FUNCTION_BLOCK FB_UMC EXTENDS FB_CtrlBase
VAR_INPUT
	In_uinStatus				: UINT;
	In_intMotorActualSpeed		: INT;
	In_uinMotorSetSpeed			: UINT;
	In_strNetId					: AMSNETID;
	In_uintPort					: WORD;
	In_uinECATState				: UINT;
	In_bolEmoOk					: BOOL;
END_VAR
VAR_OUTPUT
	Out_uinControl      	: UINT;
	Out_uinSpeedSetpoint	: UINT;
END_VAR
VAR
	/// Specific interface struct for public access
	SIf					: T_Ctrl_SIf_UMC;
	In_unStatus			: U_UMC_Lenze_Status;
	Out_unControl		: U_UMC_Lenze_Control;
	arTurnDirection		: ARRAY[0..MAX_E_TURN_DIRECTION] OF BOOL;
	fbPulse				: TC2_STANDARD.TP;
END_VAR
VAR CONSTANT
	cLEFT				: BOOL := TRUE;
	cRIGHT				: BOOL := FALSE;

	cEtherCAT_OP_MODE		: UINT := 16#0008;
	cEtherCAT_MODE_MASK		: UINT := 16#000F;
END_VAR

(*__________________________________________________________________________________________________
¦	
¦	Vistaprint Schweiz GmbH
¦	CH - 8401 Winterthur
¦
¦	www.vistaprint.ch - info@vistaprint.ch
¦___________________________________________________________________________________________________

Function desription:
Lenze Motor implementation. 


History:
Version		Date			Author		Comment
---------------------------------------------------------------------------------------------------
0.00.1		09.07.2013		PC			Start history
0.00.2		04.02.2014		AVM/MRU		Simulation mode
										cCMD_LEFT / cCMD_RIGHT added in FB_init / getCmdState

___________________________________________________________________________________________________*)


IF (me.bolActivate) THEN // cyclic call enabled
	IF (CIf.Info.bolInitDone=FALSE) THEN // first cycle -> init
		CtrlInit();
		CIf.Info.bolInitDone := TRUE;
	ELSE
		CycleStartDuty();
	
		Always();
		
		StateMachine();
		
		CycleEndDuty();
	END_IF
END_IF;

METHOD FB_init : BOOL
VAR_INPUT
	bInitRetains : BOOL; // if TRUE, the retain variables are initialized (warm start / cold start)
	bInCopyCode : BOOL;  // if TRUE, the instance afterwards gets moved into the copy code (online change)
END_VAR
VAR
	iIdx		: UINT;
	iLength		: UINT;	
END_VAR
//------------------------------------------------------------------------------------------------------------------------
// to manually change in new FUB implementation!!!
// define valid commands for this controller
iLength := SIZEOF(CIf.Job.aCmdList)/SIZEOF(CIf.Job.aCmdList[0]);
iIdx := 0;

WHILE (iIdx < iLength) AND (CIf.Job.aCmdList[iIdx].intCmd <> cCMD_INITIALIZED) DO
	iIdx := iIdx + 1; 
END_WHILE

IF (iIdx < iLength) THEN
// Add configuration of own comands	
	CIf.Job.aCmdList[iIdx].intCmd := BASE_PLC.cCMD_STOP;
	CIf.Job.aCmdList[iIdx].strName := 'Stop'; 
	CIf.Job.aCmdList[iIdx].bolAvailable := TRUE;
	iIdx := iIdx + 1;
	CIf.Job.aCmdList[iIdx].intCmd := cCMD_RUN;
	CIf.Job.aCmdList[iIdx].strName := 'Run'; 
	CIf.Job.aCmdList[iIdx].bolAvailable := TRUE;
	iIdx := iIdx + 1;
	CIf.Job.aCmdList[iIdx].intCmd := cCMD_LEFT;
	CIf.Job.aCmdList[iIdx].strName := 'Left'; 
	CIf.Job.aCmdList[iIdx].bolAvailable := TRUE;
	iIdx := iIdx + 1;
	CIf.Job.aCmdList[iIdx].intCmd := cCMD_RIGHT;
	CIf.Job.aCmdList[iIdx].strName := 'Right'; 
	CIf.Job.aCmdList[iIdx].bolAvailable := TRUE;
	iIdx := iIdx + 1;
ELSE
	;// Error if the aCmdList Array is to small
END_IF

// set name of class/typ
CIf.Info.strType := 'FB_UMC'; 

// set alarm class
SIf.Alm[E_ALM_UMC.MotorOnTimeout].eAlmClass := Base_PLC.E_AlmClass.TSTOP;
SIf.Alm[E_ALM_UMC.MotorOnTimeout].strText := 'Motor On Timeout'; 
SIf.Alm[E_ALM_UMC.MotorError].eAlmClass := Base_PLC.E_AlmClass.TSTOP;
SIf.Alm[E_ALM_UMC.MotorError].strText := 'Motor Error';
SIf.Alm[E_ALM_UMC.MotorWarning].eAlmClass := Base_PLC.E_AlmClass.WARNING;
SIf.Alm[E_ALM_UMC.MotorWarning].strText := 'Motor Warning';
SIf.Alm[E_ALM_UMC.MotorOverCurrent].eAlmClass := Base_PLC.E_AlmClass.WARNING;
SIf.Alm[E_ALM_UMC.MotorOverCurrent].strText := 'Motor Over Current';
SIf.Alm[E_ALM_UMC.MotorNotReady].eAlmClass := Base_PLC.E_AlmClass.TSTOP;
SIf.Alm[E_ALM_UMC.MotorNotReady].strText := 'Motor Not Ready';
SIf.Alm[E_ALM_UMC.DirectionParameterOverflow].eAlmClass := Base_PLC.E_AlmClass.TSTOP;
SIf.Alm[E_ALM_UMC.DirectionParameterOverflow].strText := 'Direction Parameter Overflow';
SIf.Alm[E_ALM_UMC.SpeedOverLimit].eAlmClass := Base_PLC.E_AlmClass.WARNING;
SIf.Alm[E_ALM_UMC.SpeedOverLimit].strText := 'Motor Setpoint over the limit';

//*******************************************************************************
// initial values
//*******************************************************************************

// software configuration
CIf.SwCfg.bolExist := TRUE;
CIf.SwCfg.bolEnable := TRUE;
CIf.SwCfg.bolSimulation := FALSE;

// configuration
SIf.Cfg.uinLC11 := 1500;
SIf.Cfg.uinLC11_100 := 16384;
SIf.Cfg.uinMaxSpeed := 150;

// parameter
SIf.Par.udiStartupOnTime_ms := 5000;
SIf.Par.udiMotorOnTime_ms 	:= 10000;
SIf.Par.uinSpeed_rpm 		:= 1000;
SIf.Par.uinMotorResetPulseTime_ms	:= 500;
SIf.Par.uinMotorResetCnt 		:= 3;
SIf.Par.udiMoveStartLatency 	:= 15;
SIf.Par.udiMoveStopLatency 		:= 60;
SIf.Par.eRotationDirection  := E_TURN_DIRECTION.LEFT;

SIf.Par.udiSimMotorOnTime_ms := SIf.Par.udiMotorOnTime_ms / 10;
END_METHOD

METHOD PROTECTED Always : BOOL
SUPER^.Always();

// ----------------------------------------------------------------------------------
// Simulation
IF (CIf.SwCfg.bolSimulation) THEN
	// Simulate inputs (no physical inputs)
	SIf.In.bolEmoOk.intern := TRUE;
END_IF

// ----------------------------------------------------------------------------------
// Conditions Always
IF (me.StateMachine.intState<>cSTA_SINGLE_ANSWER) THEN
	IF (((me.Alarm.eActivAlmClass=E_AlmClass.OFF) OR (me.intCmd=cCMD_OFF))
			AND (me.StateMachine.intState<>cSTA_ERROR) AND (me.StateMachine.intState<>cSTA_ERRORQuit)
			AND (me.StateMachine.intState<>cSTA_EOFF) AND (me.StateMachine.intState<>cSTA_EOFFBusy)
			AND (me.StateMachine.intState<>cSTA_OFF) AND (me.StateMachine.intState<>cSTA_OFFBusy)
			AND (me.StateMachine.intState<>UMC_CmdState.cSTA_RESETMOTORERROR) 
			AND (me.StateMachine.intState<>UMC_CmdState.cSTA_SETOPERATIONMODE)) THEN
		me.StateMachine.intStateNext := cSTA_OFFBusy;	
	END_IF

	//-------------------------------------------------------------------------------
	// Monitoring of inputs from Safety PLC (no physical inputs)
	//-------------------------------------------------------------------------------
	// Emergency Off
	IF ((SIf.In.bolEmoOk.intern = FALSE) AND (me.StateMachine.intState <> cSTA_EOFF) 
		AND (me.StateMachine.intState <> BASE_PLC.cSTA_EOFFBusy)
		AND (me.StateMachine.intState <> BASE_PLC.cSTA_ERROR) 
		AND (me.StateMachine.intState <> BASE_PLC.cSTA_PON) 
		AND (me.StateMachine.intState <> BASE_PLC.cSTA_PONBusy) 
		AND (me.StateMachine.intState<>BASE_PLC.cSTA_INITIALIZED)
		AND (me.StateMachine.intState <> BASE_PLC.cSTA_ERRORQuit)) THEN
		me.StateMachine.intStateNext := cSTA_EOFFBusy;				
	END_IF	
END_IF
END_METHOD

METHOD PROTECTED getCmdState : STRING

VAR_INPUT
	intCmdState: INT;
	bolState: BOOL;
END_VAR
getCmdState := SUPER^.getCmdState(intCmdState:=intCmdState,bolState:=bolState); // get global/base defined cmds/states

IF (getCmdState='') THEN // global not defined get local
	// get string cmd/state string information in runtime
	IF (bolState=FALSE) THEN
		// Comands's
		CASE intCmdState OF
			cCMD_LEFT: 
				getCmdState := 'cCMD_Left';
			cCMD_RIGHT: 
				getCmdState := 'cCMD_Right';
		END_CASE;
	ELSE
		// States's
		CASE intCmdState OF
			cSTA_RUN: 
				getCmdState := 'RUN';
			cSTA_RUNBusy: 
				getCmdState := 'RUNBusy';
			UMC_CmdState.cSTA_RESETMOTORERROR:
				getCmdState := 'RESETMOTORERROR';
			UMC_CmdState.cSTA_SETOPERATIONMODE:
				getCmdState := 'SETOPERATIONMODE';
		END_CASE;
	END_IF
END_IF
END_METHOD

METHOD getCtrlSIf : POINTER TO T_Ctrl_SIf_UMC
getCtrlSIf := ADR(SIf);
END_METHOD

METHOD PROTECTED IoInBridge : BOOL
// digitale and analoge inputs read from hardware or forcing
SIf.In.uinStatus.map			:= THIS^.In_uinStatus				;
SIf.In.intMotorActualSpeed.map	:= THIS^.In_intMotorActualSpeed	;
SIf.In.uinMotorSetSpeed.map		:= THIS^.In_uinMotorSetSpeed		;
SIf.In.bolEmoOk.map				:= THIS^.In_bolEmoOk		;

IF (CIf.SwCfg.bolSimulation = FALSE) THEN
	BASE_PLC.getInUint(CIf.Job.bolIoForce,ADR(SIf.In.uinStatus));
	BASE_PLC.getInUint(CIf.Job.bolIoForce,ADR(SIf.In.intMotorActualSpeed));
	BASE_PLC.getInUint(CIf.Job.bolIoForce,ADR(SIf.In.uinMotorSetSpeed));
	BASE_PLC.getInUint(CIf.Job.bolIoForce,ADR(SIf.In.bolEmoOk));
ELSE
	//simulation of global IO
END_IF
END_METHOD

METHOD PROTECTED IoOutBridge : BOOL
VAR
	bolSwitchValvesOff: BOOL;
END_VAR
// digitale and analoge inputs read from hardware or forcing
IF (CIf.SwCfg.bolSimulation = FALSE) THEN
	BASE_PLC.setOutUint(CIf.Job.bolIoForce ,ADR(SIf.Out.uinControl));
	BASE_PLC.setOutUint(CIf.Job.bolIoForce ,ADR(SIf.Out.uinSpeedSetpoint));

	THIS^.Out_uinControl			:= SIf.Out.uinControl.map	;
	THIS^.Out_uinSpeedSetpoint		:= SIf.Out.uinSpeedSetpoint.map	;
END_IF
END_METHOD

METHOD PROTECTED sta_ERROR : BOOL
// state implemetation
//--------------------------------------------------------------------------------------
// Entry action
	IF (me.StateMachine.intState<>me.StateMachine.intStateLastCycle) THEN
		me.StateMachine.intStateHistory := me.StateMachine.intStateLastCycle; // -> possibillity to go back to state before error
		me.StateMachine.intStateLastCycle := me.StateMachine.intState;
		SIf.Cur.uinMotorResetCnt := 0;
		cmd_MotorOff();
	END_IF


//--------------------------------------------------------------------------------------
// Cyclic action
	IF (me.StateMachine.intState=me.StateMachine.intStateLastCycle) THEN
		
		;
		
		
		// State Change Condition
		IF (CIf.Job.bolAlmReset = TRUE) THEN
			me.StateMachine.intStateNext := cSTA_ERRORQuit;
		END_IF
	END_IF




//--------------------------------------------------------------------------------------
// Exit action
	IF (me.StateMachine.intState<>me.StateMachine.intStateNext) THEN
		;
	END_IF
END_METHOD

METHOD PROTECTED sta_ERRORQuit : BOOL
// state implemetation
//--------------------------------------------------------------------------------------
// Entry action
	IF (me.StateMachine.intState<>me.StateMachine.intStateLastCycle) THEN
		me.StateMachine.intStateLastCycle := me.StateMachine.intState;
		
	END_IF


//--------------------------------------------------------------------------------------
// Cyclic action
	IF (me.StateMachine.intState=me.StateMachine.intStateLastCycle) THEN
		
		;
		// evtl. wait time if reset of device is necessary and then decide to go to states or ERROR state
		IF (CIf.Job.bolAlmReset = TRUE) THEN
			CIf.Job.eMe_ActivAlmClass := E_AlmClass.NONE; // reset feedback channel for parent
			CIf.Job.bolAlmReset := FALSE;
		END_IF
		
		// State Change Condition
		IF (CIf.Job.bolAlmReset = FALSE) THEN
			IF (me.StateMachine.intStateHistory<=cSTA_PON) THEN
				me.StateMachine.intStateNext := cSTA_PON;
			ELSIF (CIf.SwCfg.bolSimulation = TRUE) THEN	// Do not set operation mode in simulation
				me.StateMachine.intStateNext := BASE_PLC.cSTA_OFF;
			ELSE
				me.StateMachine.intStateNext := UMC_CmdState.cSTA_SETOPERATIONMODE;
			END_IF
		END_IF
	END_IF




//--------------------------------------------------------------------------------------
// Exit action
	IF (me.StateMachine.intState<>me.StateMachine.intStateNext) THEN
		;
	END_IF
END_METHOD

METHOD PROTECTED sta_PON : BOOL
VAR_INPUT
END_VAR
// state implemetation
//--------------------------------------------------------------------------------------
// Entry action
	IF (me.StateMachine.intState<>me.StateMachine.intStateLastCycle) THEN
		me.StateMachine.intStateLastCycle := me.StateMachine.intState;
		
	END_IF


//--------------------------------------------------------------------------------------
// Cyclic action
	IF (me.StateMachine.intState=me.StateMachine.intStateLastCycle) THEN
		;
	END_IF




//--------------------------------------------------------------------------------------
// Exit action
	IF (me.StateMachine.intState<>me.StateMachine.intStateNext) THEN
		;
	END_IF
END_METHOD

METHOD PROTECTED sta_OFFBusy : BOOL
VAR
	uinECatStatus	: UINT;
	eMotorStatus	: E_UMC_MOTOR_STATUS;
END_VAR
// state implemetation
//--------------------------------------------------------------------------------------
// Entry action
	IF (me.StateMachine.intState<>me.StateMachine.intStateLastCycle) THEN
		me.StateMachine.intStateLastCycle := me.StateMachine.intState;
		cmd_MotorOff();
	END_IF


//--------------------------------------------------------------------------------------
// Cyclic action
	IF (me.StateMachine.intState=me.StateMachine.intStateLastCycle) THEN
		eMotorStatus := GetMotorStatus(sif.In.uinStatus.intern);
		uinECatStatus := In_uinECATState AND cEtherCAT_MODE_MASK;

		IF    (uinECatStatus = cEtherCAT_OP_MODE)
		  AND NOT In_unStatus.Data.Trouble 
		  AND In_unStatus.Data.ActSpeedIsZero
		  AND (eMotorStatus = E_UMC_MOTOR_STATUS.ReadyToSwitchON) THEN
			me.StateMachine.intStateNext := Base_PLC.cSTA_OFF;
		ELSIF (CIf.SwCfg.bolSimulation = TRUE) THEN	// Do not set operation mode in simulation
			me.StateMachine.intStateNext := BASE_PLC.cSTA_OFF;
		ELSE
			IF me.StateMachine.udiTimeInState_ms > SIf.Par.uinMotorResetPulseTime_ms THEN
				IF SIf.Cur.uinMotorResetCnt > SIf.Par.uinMotorResetCnt THEN
					pfbAlarmCtrl^.setAlarm(CIf.Info.intCtrlId,INT_TO_UINT(E_ALM_UMC.MotorError),0,ADR(SIf.Alm),E_AlmState.RST,CIf.Job.eMe_ActivAlmClass);
					me.StateMachine.intStateNext := Base_PLC.cSTA_ERROR;	
				ELSE
					me.StateMachine.intStateNext := UMC_CmdState.cSTA_SETOPERATIONMODE;
				END_IF
			END_IF
		END_IF
	END_IF

//--------------------------------------------------------------------------------------
// Exit action
	IF (me.StateMachine.intState<>me.StateMachine.intStateNext) THEN
		;
	END_IF
END_METHOD

METHOD PROTECTED sta_OFF : BOOL
VAR_INPUT
END_VAR
// state implemetation
//--------------------------------------------------------------------------------------
// Entry action
	IF (me.StateMachine.intState<>me.StateMachine.intStateLastCycle) THEN
		me.StateMachine.intStateLastCycle := me.StateMachine.intState;

		SIf.Cur.uinMotorResetCnt := 0;
	END_IF


//--------------------------------------------------------------------------------------
// Cyclic action
	IF (me.StateMachine.intState=me.StateMachine.intStateLastCycle) THEN
		CASE me.intCmd OF
			cCMD_Left:
				SIf.Par.eRotationDirection := E_TURN_DIRECTION.LEFT;
				me.StateMachine.intStateNext := cSTA_RUNBusy;
			cCMD_Right:
				SIf.Par.eRotationDirection := E_TURN_DIRECTION.RIGHT;
				me.StateMachine.intStateNext := cSTA_RUNBusy;
			BASE_PLC.cCMD_STOP:
				me.StateMachine.intStateNext := BASE_PLC.cSTA_STOPBusy;
			BASE_PLC.cCMD_RUN:
				me.StateMachine.intStateNext := cSTA_RUNBusy;
		END_CASE
	END_IF


//--------------------------------------------------------------------------------------
// Exit action
	IF (me.StateMachine.intState<>me.StateMachine.intStateNext) THEN
		;
	END_IF
END_METHOD

METHOD PROTECTED StateMachine : BOOL
SUPER^.StateMachine();

// main statemachine of base controller
CASE me.StateMachine.intState OF
	cSTA_RUNBusy:
		THIS^.sta_RUNBusy();
	cSTA_RUN:
		THIS^.sta_RUN();
	cSTA_STOPBusy: 
        THIS^.sta_STOPBusy();
    cSTA_STOP: 
        THIS^.sta_STOP();
	UMC_CmdState.cSTA_RESETMOTORERROR:
		THIS^.sta_RESETMOTORERROR();
	UMC_CmdState.cSTA_SETOPERATIONMODE:
		THIS^.sta_SETOPERATIONMODE();
END_CASE;
END_METHOD

METHOD PROTECTED cmd_MotorOff : BOOL
Out_unControl.Output 				:= 0;
Out_unControl.Data.SetDCBreak 		:= 1;
Out_unControl.Data.SetHalt        	:= 1;
Out_unControl.Data.SetQuickStop    	:= 1;
SIf.Out.uinSpeedSetpoint.intern 	:= 0;
END_METHOD

METHOD PROTECTED cmd_MotorOn : BOOL
VAR_INPUT
	bDirection		: BOOL;		// Direction of the drive; False = Right; True = Left
	uinSpeed		: UINT;					// Speed of the belt
END_VAR
Out_unControl.Output 				:= 0;
Out_unControl.Data.EnableOperation 	:= 1;
Out_unControl.Data.SwitchOn        	:= 1;
Out_unControl.Data.SetSpeedCcw     	:= bDirection;

SIf.Out.uinSpeedSetpoint.intern 	:= uinSpeed;
END_METHOD

METHOD PROTECTED CycleStartDuty : BOOL
VAR_INPUT
END_VAR
SUPER^.CycleStartDuty();

In_unStatus.Input := SIf.In.uinStatus.intern;
END_METHOD

METHOD PROTECTED CycleEndDuty : BOOL
VAR_INPUT
END_VAR
SIf.Out.uinControl.intern := Out_unControl.Output;

SUPER^.CycleEndDuty();
END_METHOD

METHOD PROTECTED sta_STOPBusy : BOOL
VAR
	uniStatus 		: U_UMC_Lenze_Status;
END_VAR
// state implemetation
//--------------------------------------------------------------------------------------
// Entry action
	IF (me.StateMachine.intState<>me.StateMachine.intStateLastCycle) THEN
		me.StateMachine.intStateLastCycle := me.StateMachine.intState;
		// Switch Motor Off
		cmd_MotorStop();
	END_IF


//--------------------------------------------------------------------------------------
// Cyclic action
	IF (me.StateMachine.intState=me.StateMachine.intStateLastCycle) THEN
		IF (CIf.SwCfg.bolSimulation) THEN
			SIf.In.uinMotorSetSpeed.intern 	:= 0;
			SIf.In.intMotorActualSpeed.intern 	:= 0;
			uniStatus.Input 				:= 0;
			uniStatus.Data.ActSpeedIsZero	:= TRUE;
			SIf.In.uinStatus.intern 		:= uniStatus.Input;
		END_IF

		IF (me.StateMachine.udiTimeInState_ms < SIf.Par.udiMotorOnTime_ms) THEN
			IF (NOT In_unStatus.Data.Trouble) AND (In_unStatus.Data.ActSpeedIsZero) THEN
				me.StateMachine.intStateNext := Base_PLC.cSTA_STOP;
			END_IF;	
		ELSE
			pfbAlarmCtrl^.setAlarm(CIf.Info.intCtrlId,INT_TO_UINT(E_ALM_UMC.MotorError),0,ADR(SIf.Alm),E_AlmState.RST,CIf.Job.eMe_ActivAlmClass);
			me.StateMachine.intStateNext := Base_PLC.cSTA_ERROR;	
		END_IF
END_IF


//--------------------------------------------------------------------------------------
// Exit action
	IF (me.StateMachine.intState<>me.StateMachine.intStateNext) THEN
		Out_unControl.Data.ResetFault := FALSE;
	END_IF
END_METHOD

METHOD PROTECTED sta_STOP : BOOL
VAR_INPUT
END_VAR
// state implemetation
//--------------------------------------------------------------------------------------
// Entry action
	IF (me.StateMachine.intState<>me.StateMachine.intStateLastCycle) THEN
		me.StateMachine.intStateLastCycle := me.StateMachine.intState;

	END_IF


//--------------------------------------------------------------------------------------
// Cyclic action
	IF (me.StateMachine.intState=me.StateMachine.intStateLastCycle) THEN
		CASE me.intCmd OF
			cCMD_Left:
				SIf.Par.eRotationDirection := E_TURN_DIRECTION.LEFT;
				me.StateMachine.intStateNext := cSTA_RUNBusy;
			cCMD_Right:
				SIf.Par.eRotationDirection := E_TURN_DIRECTION.RIGHT;
				me.StateMachine.intStateNext := cSTA_RUNBusy;
			BASE_PLC.cCMD_RUN:
				me.StateMachine.intStateNext := cSTA_RUNBusy;
		END_CASE
	END_IF


//--------------------------------------------------------------------------------------
// Exit action
	IF (me.StateMachine.intState<>me.StateMachine.intStateNext) THEN
		;
	END_IF
END_METHOD

METHOD PROTECTED sta_RUNBusy : BOOL
VAR
	uniStatus 		: U_UMC_Lenze_Status;
END_VAR
// state implemetation
//--------------------------------------------------------------------------------------
// Entry action
	IF (me.StateMachine.intState<>me.StateMachine.intStateLastCycle) THEN
		me.StateMachine.intStateLastCycle := me.StateMachine.intState;

		SIf.Cur.uinSpeed_rpm := SIf.Par.uinSpeed_rpm;
		SIf.Cur.uinSpeedOuput := GetSpeedValue();
		SIf.Cur.eDirection 	:= SIf.Par.eRotationDirection;
		
		// Switch Motor ON
		IF SIf.Par.eRotationDirection < E_TURN_DIRECTION.MAX_E_TURN_DIRECTION THEN
			cmd_MotorOn(arTurnDirection[SIf.Par.eRotationDirection], SIf.Cur.uinSpeedOuput);
		ELSE
			pfbAlarmCtrl^.setAlarm(CIf.Info.intCtrlId,INT_TO_UINT(E_ALM_UMC.DirectionParameterOverflow),0,ADR(SIf.Alm),E_AlmState.RST,CIf.Job.eMe_ActivAlmClass);
			me.StateMachine.intStateNext := Base_PLC.cSTA_ERROR;	
		END_IF

		fbSimulationTimer.IN := FALSE;
		fbSimulationTimer.PT := UDINT_TO_TIME(SIf.Par.udiSimMotorOnTime_ms);
		fbSimulationTimer(); // set time/reset timer
		fbSimulationTimer.IN := TRUE; // start timer

	END_IF


//--------------------------------------------------------------------------------------
// Cyclic action
	IF (me.StateMachine.intState=me.StateMachine.intStateLastCycle) THEN
		IF (CIf.SwCfg.bolSimulation) THEN
			fbSimulationTimer(); // simulation time
			IF (fbSimulationTimer.Q) THEN
				SIf.In.uinMotorSetSpeed.intern 	:= SIf.Out.uinSpeedSetpoint.intern;
				SIf.In.uinMotorSetSpeed.intern 	:= SIf.Out.uinSpeedSetpoint.intern;
				uniStatus.Input 				:= 0;
				uniStatus.Data.DriveReady		:= 1;
				uniStatus.Data.SpeedActEqualSet := 1;
				uniStatus.Data.SpeedSetReached  := 1;
				uniStatus.Data.Status_1			:= 1;
				uniStatus.Data.Status_3			:= 1;
				uniStatus.Data.SpeedCcw			:= arTurnDirection[SIf.Par.eRotationDirection];
				SIf.In.uinStatus.intern 		:= uniStatus.Input;
			END_IF
		END_IF

		IF (me.StateMachine.udiTimeInState_ms > SIf.Par.udiMotorOnTime_ms) THEN
			pfbAlarmCtrl^.setAlarm(CIf.Info.intCtrlId,INT_TO_UINT(E_ALM_UMC.MotorOnTimeout),0,ADR(SIf.Alm),E_AlmState.RST,CIf.Job.eMe_ActivAlmClass);
			me.StateMachine.intStateNext := Base_PLC.cSTA_ERROR;	
		END_IF

		IF In_unStatus.Data.Trouble THEN
			pfbAlarmCtrl^.setAlarm(CIf.Info.intCtrlId,INT_TO_UINT(E_ALM_UMC.MotorError),0,ADR(SIf.Alm),E_AlmState.RST,CIf.Job.eMe_ActivAlmClass);
			me.StateMachine.intStateNext := Base_PLC.cSTA_ERROR;	
		END_IF
		
		IF (me.StateMachine.intStateNext <> Base_PLC.cSTA_ERROR) THEN
			IF (NOT In_unStatus.Data.Trouble) 
				AND (THIS^.arTurnDirection[SIf.Cur.eDirection] = In_unStatus.Data.SpeedCcw)	THEN
//				AND (In_unStatus.Data.SpeedSetReached) THEN
				me.StateMachine.intStateNext := cSTA_RUN;
			END_IF;	

			// Reenter the RunBusy state again if the speed changes
			IF GetSpeedValue() <> SIf.Cur.uinSpeedOuput THEN
				me.StateMachine.intStateLastCycle := -1;
			END_IF
			
			// Reenter the RunBusy state again if the direction changes.
			IF SIf.Par.eRotationDirection <> SIf.Cur.eDirection THEN
				me.StateMachine.intStateLastCycle := -1;
			END_IF
			
			CASE me.intCmd OF
				cCMD_Left:
					IF SIf.Par.eRotationDirection <> E_TURN_DIRECTION.LEFT THEN
						SIf.Par.eRotationDirection := E_TURN_DIRECTION.LEFT;
						me.StateMachine.intStateLastCycle := -1;
					END_IF
				cCMD_Right:
					IF SIf.Par.eRotationDirection <> E_TURN_DIRECTION.RIGHT THEN
						SIf.Par.eRotationDirection := E_TURN_DIRECTION.RIGHT;
						me.StateMachine.intStateLastCycle := -1;
					END_IF
				BASE_PLC.cCMD_STOP:
					me.StateMachine.intStateNext := BASE_PLC.cSTA_STOPBusy;
			END_CASE
		END_IF
END_IF


//--------------------------------------------------------------------------------------
// Exit action
	IF (me.StateMachine.intState<>me.StateMachine.intStateNext) THEN
		;
	END_IF
END_METHOD

METHOD PROTECTED sta_RUN : BOOL
VAR
	uniStatus 		: U_UMC_Lenze_Status;
END_VAR
// state implemetation
//--------------------------------------------------------------------------------------
// Entry action
	IF (me.StateMachine.intState<>me.StateMachine.intStateLastCycle) THEN
		me.StateMachine.intStateLastCycle := me.StateMachine.intState;
		CIf.Job.intACmd := BASE_PLC.cCMD_DONE;
	END_IF


//--------------------------------------------------------------------------------------
// Cyclic action
	IF (me.StateMachine.intState=me.StateMachine.intStateLastCycle) THEN
		IF In_unStatus.Data.Trouble THEN
			pfbAlarmCtrl^.setAlarm(CIf.Info.intCtrlId,INT_TO_UINT(E_ALM_UMC.MotorError),0,ADR(SIf.Alm),E_AlmState.RST,CIf.Job.eMe_ActivAlmClass);
			me.StateMachine.intStateNext := Base_PLC.cSTA_ERROR;	
		END_IF
		
		IF (me.StateMachine.intStateNext <> Base_PLC.cSTA_ERROR) THEN
			// Reenter the RunBusy state again if the speed changes
			IF SIf.Par.uinSpeed_rpm <> SIf.Cur.uinSpeed_rpm THEN
				me.StateMachine.intStateNext := cSTA_RUNBusy;
			END_IF
			
			// Reenter the RunBusy state again if the direction changes.
			IF SIf.Par.eRotationDirection <> SIf.Cur.eDirection THEN
				me.StateMachine.intStateNext := cSTA_RUNBusy;
			END_IF

			CASE me.intCmd OF
				cCMD_Left:
					SIf.Par.eRotationDirection := E_TURN_DIRECTION.LEFT;
					me.StateMachine.intStateNext := cSTA_RUNBusy;
				cCMD_Right:
					SIf.Par.eRotationDirection := E_TURN_DIRECTION.RIGHT;
					me.StateMachine.intStateNext := cSTA_RUNBusy;
				BASE_PLC.cCMD_STOP:
					me.StateMachine.intStateNext := BASE_PLC.cSTA_STOPBusy;
			END_CASE
		END_IF
END_IF


//--------------------------------------------------------------------------------------
// Exit action
	IF (me.StateMachine.intState<>me.StateMachine.intStateNext) THEN
		;
	END_IF
END_METHOD

METHOD PROTECTED CtrlInit : BOOL
VAR_INPUT
END_VAR
SUPER^.CtrlInit();

arTurnDirection[E_TURN_DIRECTION.AUTOMATIC] := FALSE;
arTurnDirection[E_TURN_DIRECTION.LEFT] 		:= FALSE;
arTurnDirection[E_TURN_DIRECTION.RIGHT] 	:= TRUE;

SIf.Cur.uinSpeedLimit := SIf.Cfg.uinMaxSpeed * SIf.Cfg.uinLC11_100 / 100;
END_METHOD

METHOD PROTECTED GetSpeedValue : UINT
VAR
	uinSpeedOutput			: UINT;
END_VAR
uinSpeedOutput := SIf.Par.uinSpeed_rpm * SIf.Cfg.uinLC11_100 / SIf.Cfg.uinLC11;

IF uinSpeedOutput > SIf.Cur.uinSpeedLimit THEN
	uinSpeedOutput := SIf.Cur.uinSpeedLimit;
	pfbAlarmCtrl^.setAlarm(CIf.Info.intCtrlId,INT_TO_UINT(E_ALM_UMC.SpeedOverLimit),0,ADR(SIf.Alm),E_AlmState.RST,CIf.Job.eMe_ActivAlmClass);
END_IF

GetSpeedValue := uinSpeedOutput;
END_METHOD

METHOD PROTECTED cmd_MotorReset : BOOL
VAR_INPUT
END_VAR
cmd_MotorOff();
Out_unControl.Data.ResetFault 		:= 1;
END_METHOD

METHOD PROTECTED GetMotorStatus : E_UMC_MOTOR_STATUS
VAR_INPUT
	uinMotorStatus		: UINT;
END_VAR
uinMotorStatus := uinMotorStatus AND 16#0F00;
uinMotorStatus := SHR(uinMotorStatus,8);
GetMotorStatus := UINT_TO_INT(uinMotorStatus);
END_METHOD

METHOD PROTECTED cmd_MotorStop : BOOL
VAR_INPUT
END_VAR
Out_unControl.Output 				:= 0;
Out_unControl.Data.SetDCBreak 		:= 1;
Out_unControl.Data.SetHalt        	:= 1;
Out_unControl.Data.SetQuickStop    	:= 1;
END_METHOD

METHOD PROTECTED sta_SETOPERATIONMODE : BOOL
VAR
	uinECatStatus		: UINT;

	fbEcReqSlaveState 	: FB_EcReqSlaveState;
	bExecute        	: BOOL;
	uinReqState     	: WORD := EC_DEVICE_STATE_OP;
	bError          	: BOOL;
	nErrId          	: UDINT;
END_VAR
// state implemetation
//--------------------------------------------------------------------------------------
// Entry action
	IF (me.StateMachine.intState<>me.StateMachine.intStateLastCycle) THEN
		me.StateMachine.intStateLastCycle := me.StateMachine.intState;
	END_IF


//--------------------------------------------------------------------------------------
// Cyclic action
	IF (me.StateMachine.intState=me.StateMachine.intStateLastCycle) THEN
		bExecute := NOT ((In_uinECATState AND cEtherCAT_MODE_MASK) = cEtherCAT_OP_MODE);

		IF NOT bExecute THEN
			me.StateMachine.intStateNext := UMC_CmdState.cSTA_RESETMOTORERROR;
		END_IF

		fbEcReqSlaveState(
			sNetId		:= F_CreateAmsNetId(In_strNetId), 
			nSlaveAddr	:= In_uintPort, 
			bExecute	:= bExecute, 
			state		:= uinReqState  );

		IF (me.StateMachine.udiTimeInState_ms > SIf.Par.udiStartupOnTime_ms) THEN
			pfbAlarmCtrl^.setAlarm(CIf.Info.intCtrlId,INT_TO_UINT(E_ALM_UMC.MotorError),0,ADR(SIf.Alm),E_AlmState.RST,CIf.Job.eMe_ActivAlmClass);
			me.StateMachine.intStateNext := Base_PLC.cSTA_ERROR;	
		END_IF
END_IF


//--------------------------------------------------------------------------------------
// Exit action
	IF (me.StateMachine.intState<>me.StateMachine.intStateNext) THEN
		Out_unControl.Data.ResetFault := FALSE;
	END_IF
END_METHOD

METHOD PROTECTED sta_RESETMOTORERROR : BOOL
VAR
	eMotorStatus	: E_UMC_MOTOR_STATUS;
END_VAR
// state implemetation
//--------------------------------------------------------------------------------------
// Entry action
	IF (me.StateMachine.intState<>me.StateMachine.intStateLastCycle) THEN
		me.StateMachine.intStateLastCycle := me.StateMachine.intState;
		cmd_MotorReset();
	END_IF


//--------------------------------------------------------------------------------------
// Cyclic action
	IF (me.StateMachine.intState=me.StateMachine.intStateLastCycle) THEN
		eMotorStatus := GetMotorStatus(sif.In.uinStatus.intern);

		IF me.SubStateMachine.udiTimeInState_ms > SIf.Par.uinMotorResetPulseTime_ms THEN
			SIf.Cur.uinMotorResetCnt := SIf.Cur.uinMotorResetCnt + 1;
			me.StateMachine.intStateNext := BASE_PLC.cSTA_OFFBusy;
		END_IF
	END_IF


//--------------------------------------------------------------------------------------
// Exit action
	IF (me.StateMachine.intState<>me.StateMachine.intStateNext) THEN
		Out_unControl.Data.ResetFault := FALSE;
	END_IF
END_METHOD

METHOD PROTECTED sta_EOFF : BOOL
VAR_INPUT
END_VAR
// state implemetation
//--------------------------------------------------------------------------------------
// Entry action
	IF (me.StateMachine.intState<>me.StateMachine.intStateLastCycle) THEN
		me.StateMachine.intStateLastCycle := me.StateMachine.intState;	
	END_IF

//--------------------------------------------------------------------------------------
// Cyclic action
	IF (me.StateMachine.intState=me.StateMachine.intStateLastCycle) THEN		
		// As long as the EMO is not reseted!
		IF SIf.In.bolEmoOk.intern THEN
			me.StateMachine.intStateNext := BASE_PLC.cSTA_OFFBusy;			
		ELSE
			IF me.intCmd <> BASE_PLC.cCMD_OFF THEN
				// Clear pending and new commands cyclic to prevent automatic recovery!	
				CIf.Job.intACmd := BASE_PLC.cCMD_DONE;
				CIf.Job.intMCmd := BASE_PLC.cCMD_DONE;		
			END_IF
		END_IF
	END_IF

//--------------------------------------------------------------------------------------
// Exit action
	IF (me.StateMachine.intState<>me.StateMachine.intStateNext) THEN
		;
	END_IF
END_METHOD

METHOD PROTECTED sta_EOFFbusy : BOOL
VAR_INPUT
END_VAR
// state implemetation
//--------------------------------------------------------------------------------------
// Entry action
IF (me.StateMachine.intState<>me.StateMachine.intStateLastCycle) THEN
	me.StateMachine.intStateLastCycle := me.StateMachine.intState;
	cmd_MotorOff();
END_IF

//--------------------------------------------------------------------------------------
// Cyclic action
IF (me.StateMachine.intState=me.StateMachine.intStateLastCycle) THEN
	IF (TRUE) THEN
		me.StateMachine.intStateNext := BASE_PLC.cSTA_EOFF;
	END_IF
END_IF

//--------------------------------------------------------------------------------------
// Exit action
IF (me.StateMachine.intState<>me.StateMachine.intStateNext) THEN
	;
END_IF
END_METHOD

PROPERTY PUBLIC CtrlSIf : POINTER TO T_Ctrl_SIf_UMC
GET
CtrlSIf := ADR(SIf);
END_GET
SET
END_SET
END_PROPERTY

END_FUNCTION_BLOCK

(* stored: Version 1.1.0.1, ProductVersion 3.1.0.19
   POU FB_UMC: Id {95b426bb-96dc-4ca4-9df1-b53c93e4707b}
   Method FB_init: Id {a745ae60-38a1-42bf-9cab-5742f75b9766}
   Method Always: Id {47fa4c02-141a-44a5-9bd0-72272f1d4112}
   Method getCmdState: Id {142cba6f-071e-4fbc-9b2e-8f6d03c2b875}
   Method getCtrlSIf: Id {acb56b64-0a6e-4c07-93ae-4c4905c668b4}
   Method IoInBridge: Id {e96c8918-614f-4a10-b14d-7ccad3e92fa6}
   Method IoOutBridge: Id {d1f368f7-6114-4b3a-a3b7-893a4112fcc7}
   Method sta_ERROR: Id {81678cf7-d126-4a6f-b2e1-afa2645116d6}
   Method sta_ERRORQuit: Id {4ff591d5-1166-4edf-964c-9bb76285ccb4}
   Method sta_PON: Id {2311706f-676b-4db4-9141-5b41e21fa6e7}
   Method sta_OFFBusy: Id {d535dac6-29f0-4c66-a808-4d4fa368fe03}
   Method sta_OFF: Id {90f727a3-208a-41ee-8fa0-865956879137}
   Method StateMachine: Id {b02dbe36-1201-40e8-9b9c-9bb09d9c998c}
   Method cmd_MotorOff: Id {20537daa-c4c1-4fa9-a96c-810bc92e7ace}
   Method cmd_MotorOn: Id {5fba66c0-ff72-4abf-a6cf-a878375ce832}
   Method CycleStartDuty: Id {52dc840d-ed8a-4517-af3d-9d0805703d2b}
   Method CycleEndDuty: Id {be820387-c131-49cd-8a3e-ec5c466b2768}
   Method sta_STOPBusy: Id {b55f6f1f-e285-4e9b-87d3-20b9bd30135c}
   Method sta_STOP: Id {fabf4a40-db3a-455c-9e73-b959fe6544f7}
   Method sta_RUNBusy: Id {5677b46f-6b90-4f51-8f06-07809321a849}
   Method sta_RUN: Id {ca1f6dc3-8b4a-4f81-a2ec-bc79c70cea58}
   Method CtrlInit: Id {3d6278bc-4119-4d76-a46c-9220dc78a04c}
   Method GetSpeedValue: Id {8377784a-78d3-4660-ba1c-318606b30ca3}
   Method cmd_MotorReset: Id {efe6cd65-958e-40ee-a863-1c37135f956e}
   Method GetMotorStatus: Id {79c8cc2d-da91-4664-bef0-d7010296b689}
   Method cmd_MotorStop: Id {152850e5-84a6-4d14-9e9c-c0b18ab6dc05}
   Method sta_SETOPERATIONMODE: Id {6e71e2b6-44ba-4353-ae18-ab8e79f0c705}
   Method sta_RESETMOTORERROR: Id {c4bd1966-3b93-4b08-9e75-20f93b303fe1}
   Method sta_EOFF: Id {517d1816-ab01-4702-9554-90bf346088dc}
   Method sta_EOFFbusy: Id {a0e681a9-b1a0-4235-80d7-2d11be64d287}
   Property CtrlSIf: Id {647335bc-e279-4764-9976-06282d07dd64}
   Get Get: Id {00c3feb1-2e98-444a-b023-2a28f641132d}
   Set Set: Id {73ee206d-060a-4c20-94b1-47268f2dbfb6} *)
